VISUALIZATION Model  // 920x568
END_VISUALIZATION

(* stored: Version 1.1.0.1
   Visu Model: Id {1ad760d6-49f5-452c-b8f8-8c412b5e472d} *)
